// SIMATIC S7-200 project (STEP 7-Micro/WIN), CPU 224XP REL 02.01

SYMBOL_TABLE USER1
start            I0.0     // khoi dong
stopp            I0.1     // dung khan cap
s1               I0.2     // cam bien hop
s2               I0.3     // cam bien dem qua
k1               Q0.0     // bang chuyen hop
k2               Q0.1     // bang chuyen qua
END_SYMBOL_TABLE

ORGANIZATION_BLOCK MAIN:OB1
TITLE=PROGRAM COMMENTS
BEGIN
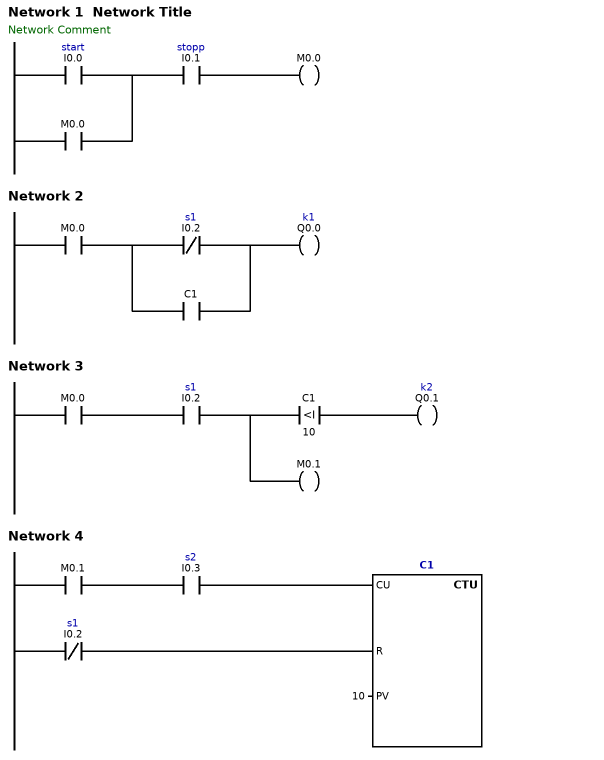
Network 1 // Network Title
// Network Comment
LD     start:I0.0
O      M0.0
A      stopp:I0.1
=      M0.0
Network 2
LD     M0.0
LDN    s1:I0.2
O      C1
ALD
=      k1:Q0.0
Network 3
LD     M0.0
A      s1:I0.2
LPS
AW<    C1, 10
=      k2:Q0.1
LPP
=      M0.1
Network 4
// (network saved uncompiled; LAD cells follow)
// row 0: c0 -| |- M0.1  c1 -| |- s2:I0.3  c2 --  c3 [CTU C1 CU:=power@row0, R:=power@row1, PV:=10]
// row 1: c0 -|/|- s1:I0.2  c1 --  c2 --  c3 [box]
// row 2: c3 [box]
END_ORGANIZATION_BLOCK
